FUNCTION_BLOCK SonotecFreq
VAR_INPUT
	rawCount  AT %I* : UDINT;
	scale : sEU_SCALE := (rawLo := 0, rawHi := 20, euLo := -20.0,  euHi := 500.0, eu := 'ml/min');
END_VAR
VAR_OUTPUT
	pv : LREAL;
END_VAR
VAR
	lastCount : UDINT := 0;
	thisCount : INT;
END_VAR

thisCount := UDINT_TO_INT(rawCount - lastCount);
lastcount := rawCount;

SonotecFreq.pv := scale.euLo + (thisCount - scale.rawLo)*(scale.euHi - scale.euLo)/(scale.rawHi - scale.rawLo);

END_FUNCTION_BLOCK

(* stored: Version 1.1.0.1, ProductVersion 3.1.0.36
   POU SonotecFreq: Id {cf3cb695-b8a6-4748-9967-bdd46f426900}, SpecialFunc None *)
